Staubli VAL3: AfterOpenLaser.pgx

public program AfterOpenLaser(num x_nWorkplaceIn, num x_nTrajIndex)
begin
  //参数：x_nWorkplaceIn 工位序号，传入的参数是 DataBase:nWorkPlaceIndex
  //参数：x_nTrajIndex 路径序号，传入的参数是TxtFile:nReadTrajIndex
  //引用位置:Motion:Move.pgx
  //功能：激光打开以后需要做的动作
  //备注：机械手臂在穿孔的时候






end
